// TwinCAT 3 PLC project PLC_Project
// ProgramVersion: 3.1.4024.0
// libraries:
//   Tc2_MC2, * (Beckhoff Automation GmbH)
//   Tc2_Standard, * (Beckhoff Automation GmbH)
//   Tc2_System, * (Beckhoff Automation GmbH)
//   Tc3_Module, * (Beckhoff Automation GmbH)
//   VisuSymbols,3.5.10.0,System
// project tree:
//   / GlobalTextList.TcGTLO, PlcTask.TcTTO, Visualization Manager.TcVMO (not stored), VISU_TASK.TcTTO
//   GVLs/ GVL_VARS1.TcGVL, GVL_VARS2.TcGVL, GVL_VARS3.TcGVL, GVL_VARS4.TcGVL
//   POUs/ FB_Functions.TcPOU, MAIN.TcPOU
//   VISUs/ Screen1.TcVIS
// real-time tasks:
//   TASK PlcTask: cycle T#10ms, priority 20, ADS port 350
//   TASK VISU_TASK: cycle T#200000us, priority 30, ADS port 351
// motion (NC):
//   TASK NC-Project1 SAF: cycle T#2ms, priority 4, ADS port 501
//   TASK NC-Project1 SVB: cycle T#10ms, priority 8, ADS port 511
//   AXIS Axis 1 (id 1)
//     OtherSettings: AllowMotionCmdToSlave=true
//     encoder EncType=1
//     encoder EncId=129, EncType=1
//     drive DrvType=5
//       Analog: TorqueSetpointScale=10, ScaleFactorActTorque=0.1
//       TimeComp: TaskDelayCycles=1
//     controller CtrType=1
//       CtrPara: PriorControlFactor=1
//         Observer: BandWidth=20
//     controller CtrId=129, CtrType=1
//       CtrPara: PriorControlFactor=1
//         Observer: BandWidth=20
//   AXIS Axis 2 (id 2)
//     OtherSettings: AllowMotionCmdToSlave=true
//     encoder EncType=1
//     encoder EncId=130, EncType=1
//     drive DrvType=5
//       Analog: TorqueSetpointScale=10, ScaleFactorActTorque=0.1
//       TimeComp: TaskDelayCycles=1
//     controller CtrType=1
//       CtrPara: PriorControlFactor=1
//         Observer: BandWidth=20
//     controller CtrId=130, CtrType=1
//       CtrPara: PriorControlFactor=1
//         Observer: BandWidth=20
//   AXIS Axis 3 (id 3)
//     OtherSettings: AllowMotionCmdToSlave=true
//     encoder EncType=1
//     encoder EncId=131, EncType=1
//     drive DrvType=5
//       Analog: TorqueSetpointScale=10, ScaleFactorActTorque=0.1
//       TimeComp: TaskDelayCycles=1
//     controller CtrType=1
//       CtrPara: PriorControlFactor=1
//         Observer: BandWidth=20
//     controller CtrId=131, CtrType=1
//       CtrPara: PriorControlFactor=1
//         Observer: BandWidth=20
//   AXIS Axis 4 (id 4)
//     OtherSettings: AllowMotionCmdToSlave=true
//     encoder EncType=1
//     encoder EncId=132, EncType=1
//     drive DrvType=5
//       Analog: TorqueSetpointScale=10, ScaleFactorActTorque=0.1
//       TimeComp: TaskDelayCycles=1
//     controller CtrType=1
//       CtrPara: PriorControlFactor=1
//         Observer: BandWidth=20
//     controller CtrId=132, CtrType=1
//       CtrPara: PriorControlFactor=1
//         Observer: BandWidth=20
// variable links:
//   PLC-Project/PLC-Project Instance <-> NC-Project1 SAF/Axes/Axis 1
//     PlcTask Inputs/MAIN.Axis[0][0].NcToPlc <-> Outputs/ToPlc
//     PlcTask Inputs/MAIN.Axis[0][1].NcToPlc <-> Outputs/ToPlc2
//     PlcTask Outputs/MAIN.Axis[0][0].PlcToNc <-> Inputs/FromPlc
//     PlcTask Outputs/MAIN.Axis[0][1].PlcToNc <-> Inputs/FromPlc2
//   PLC-Project/PLC-Project Instance <-> NC-Project1 SAF/Axes/Axis 2
//     PlcTask Inputs/MAIN.Axis[1][0].NcToPlc <-> Outputs/ToPlc
//     PlcTask Inputs/MAIN.Axis[1][1].NcToPlc <-> Outputs/ToPlc2
//     PlcTask Outputs/MAIN.Axis[1][0].PlcToNc <-> Inputs/FromPlc
//     PlcTask Outputs/MAIN.Axis[1][1].PlcToNc <-> Inputs/FromPlc2
//   PLC-Project/PLC-Project Instance <-> NC-Project1 SAF/Axes/Axis 3
//     PlcTask Inputs/MAIN.Axis[2][0].NcToPlc <-> Outputs/ToPlc
//     PlcTask Inputs/MAIN.Axis[2][1].NcToPlc <-> Outputs/ToPlc2
//     PlcTask Outputs/MAIN.Axis[2][0].PlcToNc <-> Inputs/FromPlc
//     PlcTask Outputs/MAIN.Axis[2][1].PlcToNc <-> Inputs/FromPlc2
//   PLC-Project/PLC-Project Instance <-> NC-Project1 SAF/Axes/Axis 4
//     PlcTask Inputs/MAIN.Axis[3][0].NcToPlc <-> Outputs/ToPlc
//     PlcTask Inputs/MAIN.Axis[3][1].NcToPlc <-> Outputs/ToPlc2
//     PlcTask Outputs/MAIN.Axis[3][0].PlcToNc <-> Inputs/FromPlc
//     PlcTask Outputs/MAIN.Axis[3][1].PlcToNc <-> Inputs/FromPlc2

CONFIGURATION PLC_Project
    RESOURCE PLC ON TwinCAT3
        TASK PlcTask(INTERVAL := T#10ms, PRIORITY := 20);
        TASK VISU_TASK(INTERVAL := T#200000us, PRIORITY := 30);
        PROGRAM MAIN WITH PlcTask : MAIN;
        PROGRAM VisuElems_Visu_Prg WITH VISU_TASK : VisuElems.Visu_Prg;
    END_RESOURCE
END_CONFIGURATION

// ---- GVLs/GVL_VARS1.TcGVL
{attribute 'qualified_only'}
VAR_GLOBAL
	position: UINT := 0;
	velocity: UINT := 0;
	acceleration: UINT := 0;
	execute: BOOL := FALSE;
END_VAR

// ---- GVLs/GVL_VARS2.TcGVL
{attribute 'qualified_only'}
VAR_GLOBAL
	position: UINT := 0;
	velocity: UINT := 0;
	acceleration: UINT := 0;
	execute: BOOL := FALSE;
END_VAR

// ---- GVLs/GVL_VARS3.TcGVL
{attribute 'qualified_only'}
VAR_GLOBAL
	position: UINT := 0;
	velocity: UINT := 0;
	acceleration: UINT := 0;
	execute: BOOL := FALSE;
END_VAR

// ---- GVLs/GVL_VARS4.TcGVL
{attribute 'qualified_only'}
VAR_GLOBAL
	position: UINT := 0;
	velocity: UINT := 0;
	acceleration: UINT := 0;
	execute: BOOL := FALSE;
END_VAR

// ---- POUs/MAIN.TcPOU
PROGRAM MAIN
VAR
	//nState: UINT := 0;
	Axis : ARRAY [0..3] OF ARRAY [0..1] OF AXIS_REF;
	MoveAbsolute : MC_MoveAbsolute;
	MoveRelative : MC_MoveRelative;
	WriteParameter : MC_WriteParameter;
	ReadParameter : MC_ReadParameter;
	AxisPower : MC_Power;
	Reset : MC_Reset;
	FB_Functions : FB_Functions;
	AxisParams : MC_AxisParameter;
	ReadDriveAddress : MC_ReadDriveAddress;
	SetControlLoop : MC_SelectControlLoop;
	ReadBoolParameter : MC_ReadBoolParameter;
	WriteBoolParameter : MC_WriteBoolParameter;
	Axis1LoopID : UINT;
	Axis2LoopID : UINT;
	Axis3LoopID : UINT;
	Axis4LoopID : UINT;
END_VAR

//Axis1[0]();
//Axis1[1]();
//Axis1[2]();
//Axis1();

Axis[0][0](); // incremental encoder axis 1
Axis[0][1](); // absolute encoder axis 1
Axis1LoopID := Axis[0][0].NcToPlc.ActiveControlLoopIndex;

Axis[1][0](); // incremental encoder axis 2
Axis[1][1](); // absolute encoder axis 2
Axis2LoopID := Axis[1][0].NcToPlc.ActiveControlLoopIndex;

Axis[2][0](); // incremental encoder axis 3
Axis[2][1](); // absolute encoder axis 3
Axis3LoopID := Axis[2][0].NcToPlc.ActiveControlLoopIndex;

Axis[3][0](); // incremental encoder axis 4
Axis[3][1](); // absolute encoder axis 4
Axis4LoopID := Axis[3][0].NcToPlc.ActiveControlLoopIndex;



//E_NcEncoderType.NcEncoderType_Simulation

//CASE nState OF
//	0:
//	nState := 10;
//	
//	10:
//	MoveAbsolute(Axis:=Axis1[0],Execute:=FALSE);
//	Reset(Axis:=Axis1[0],Execute:=FALSE);
//	nState := 20;
//	
//	20:
//	AxisPower(Axis:=Axis1[0],
//			Enable:=TRUE,
//			Enable_Positive:=TRUE,
//			Enable_Negative:=TRUE);
//			
//	IF GVL_VARS1.execute THEN
//		nState := 30;
//	END_IF
//
//	
//	30:
//	MoveAbsolute(Axis:=Axis1[0],
//					Position:=GVL_VARS1.position,
//					Velocity:=GVL_VARS1.velocity);
//	MoveAbsolute(Axis:=Axis1[0],
//					Execute:=TRUE);		
//	IF MoveAbsolute.Done THEN
//		MoveAbsolute(Axis:=Axis1[0],Execute:=FALSE);
//	END_IF
//	GVL_VARS1.execute := FALSE;
//	nState := 10;
//END_CASE


//AxisPower(Axis:=Axis1);
//MoveAbsolute(Axis:=Axis1);
//Reset(Axis:=Axis1);

END_PROGRAM

// ---- POUs/FB_Functions.TcPOU
FUNCTION_BLOCK FB_Functions
VAR_INPUT
END_VAR
VAR_OUTPUT
END_VAR
VAR
END_VAR

{attribute 'TcRpcEnable'}
METHOD M_EnableAxis : BOOL
VAR_INPUT
	axisID : UINT;
	loopID : UINT;
END_VAR
Main.AxisPower(Axis:=Main.Axis[axisID][loopID],Enable:=TRUE,Enable_Positive:=TRUE,Enable_Negative:=TRUE); 

RETURN;
END_METHOD

{attribute 'TcRpcEnable'}
METHOD M_MoveAbsolute : BOOL
VAR_INPUT
	axisID : UINT;
	loopID : UINT;
	position : LREAL;
	velocity : LREAL;
END_VAR
Main.AxisPower(Axis:=Main.Axis[axisID][loopID],Enable:=TRUE,Enable_Positive:=TRUE,Enable_Negative:=TRUE); 

WHILE Main.Axis[axisID][loopID].Status.Operational = FALSE DO
	Main.MoveAbsolute(Axis:=Main.Axis[axisID][loopID],Execute:=FALSE);
END_WHILE

Main.MoveAbsolute(Axis:=Main.Axis[axisID][loopID],Execute:=FALSE);
Main.Reset(Axis:=Main.Axis[axisID][loopID],Execute:=FALSE);
			
Main.MoveAbsolute(Axis:=main.Axis[axisID][loopID],Position:=position,Velocity:=velocity);
					
Main.MoveAbsolute(Axis:=Main.Axis[axisID][loopID],Execute:=TRUE);

Main.MoveAbsolute(Axis:=Main.Axis[axisID][loopID],Execute:=FALSE);

RETURN;
END_METHOD

{attribute 'TcRpcEnable'}
METHOD M_MoveHome : BOOL
VAR_INPUT
	axisID : UINT;
	loopID : UINT;
END_VAR
Main.AxisPower(Axis:=Main.Axis[axisID][loopID],Enable:=TRUE,Enable_Positive:=TRUE,Enable_Negative:=TRUE); 

WHILE Main.Axis[axisID][loopID].Status.Operational = FALSE DO
	Main.MoveHome(Axis:=Main.Axis[axisID][loopID],Execute:=FALSE);
END_WHILE

Main.MoveHome(Axis:=Main.Axis[axisID][loopID],Execute:=FALSE);
Main.Reset(Axis:=Main.Axis[axisID][loopID],Execute:=FALSE);

Main.MoveHome(Axis:=Main.Axis[axisID][loopID],Position:=0,HomingMode:=MC_DefaultHoming);

Main.MoveHome(Axis:=Main.Axis[axisID][loopID],Execute:=TRUE);

RETURN;
END_METHOD

{attribute 'TcRpcEnable'}
METHOD M_MoveRelative : BOOL
VAR_INPUT
	axisID : UINT;
	loopID : UINT;
	position : LREAL;
	velocity : LREAL;
END_VAR
Main.AxisPower(Axis:=Main.Axis[axisID][loopID],Enable:=TRUE,Enable_Positive:=TRUE,Enable_Negative:=TRUE); 

WHILE Main.Axis[axisID][loopID].Status.Operational = FALSE DO
	Main.MoveRelative(Axis:=Main.Axis[axisID][loopID],Execute:=FALSE);
END_WHILE

Main.MoveRelative(Axis:=Main.Axis[axisID][loopID],Execute:=FALSE);
Main.Reset(Axis:=Main.Axis[axisID][loopID],Execute:=FALSE);
			
Main.MoveRelative(Axis:=Main.Axis[axisID][loopID],Distance:=position,Velocity:=velocity);
					
Main.MoveRelative(Axis:=Main.Axis[axisID][loopID],Execute:=TRUE);

Main.MoveRelative(Axis:=Main.Axis[axisID][loopID],Execute:=FALSE);

RETURN;
END_METHOD

{attribute 'TcRpcEnable'}
METHOD M_ReadActiveLoop : UINT
VAR_INPUT
	axisID : UINT;
END_VAR
VAR_OUTPUT
	loopID : UINT;
END_VAR
loopID := Main.Axis[axisID][0].NcToPlc.ActiveControlLoopIndex;

RETURN;
END_METHOD

{attribute 'TcRpcEnable'}
METHOD M_ReadAxisMotion : LREAL
VAR_INPUT
	axisID : UINT;
END_VAR
VAR_OUTPUT
	position : LREAL;
	velocity : LREAL;
END_VAR
position := Main.Axis[axisID][0].NcToPlc.ActPos;

velocity := MAIN.Axis[axisID][0].NcToPlc.ActVelo;
END_METHOD

{attribute 'TcRpcEnable'}
METHOD M_ReadAxisParameters : LREAL
VAR_INPUT
	axisID : UINT;
	loopID : UINT;
END_VAR
VAR_OUTPUT
	maxVelocity : LREAL;
	maxAcceleration : LREAL;
	defaultAcceleration : LREAL;
	defaultJerk : LREAL;
	homingVelocity : LREAL;
	manualVelocityFast : LREAL;
	manualVelocitySlow : LREAL;
	jogIncrement : LREAL;
END_VAR
// Axis Max Velocity
Main.ReadParameter(Axis:=Main.Axis[axisID][loopID],ParameterNumber:=MC_AxisParameter.AxisMaxVelocity);
Main.ReadParameter(Axis:=Main.Axis[axisID][loopID],Enable:=TRUE);
WHILE Main.ReadParameter.Busy DO
	Main.ReadParameter(Axis:=Main.Axis[axisID][loopID],Enable:=FALSE);
END_WHILE
maxVelocity := Main.ReadParameter.Value;


// Axis Max Acceleration
Main.ReadParameter(Axis:=Main.Axis[axisID][loopID],ParameterNumber:=MC_AxisParameter.AxisMaximumAcceleration);
Main.ReadParameter(Axis:=Main.Axis[axisID][loopID],Enable:=TRUE);
WHILE Main.ReadParameter.Busy DO
	Main.ReadParameter(Axis:=Main.Axis[axisID][loopID],Enable:=FALSE);
END_WHILE
maxAcceleration := Main.ReadParameter.Value;


//Axis Default Acceleration
Main.ReadParameter(Axis:=Main.Axis[axisID][loopID],ParameterNumber:=MC_AxisParameter.AxisAcc);
Main.ReadParameter(Axis:=Main.Axis[axisID][loopID],Enable:=TRUE);
WHILE Main.ReadParameter.Busy DO
	Main.ReadParameter(Axis:=Main.Axis[axisID][loopID],Enable:=FALSE);
END_WHILE
defaultAcceleration := Main.ReadParameter.Value;


//Axis Default Jerk
Main.ReadParameter(Axis:=Main.Axis[axisID][loopID],ParameterNumber:=MC_AxisParameter.AxisJerk);
Main.ReadParameter(Axis:=Main.Axis[axisID][loopID],Enable:=TRUE);
WHILE Main.ReadParameter.Busy DO
	Main.ReadParameter(Axis:=Main.Axis[axisID][loopID],Enable:=FALSE);
END_WHILE
defaultJerk := Main.ReadParameter.Value;


//Axis Homing Velocity +ve direction
Main.ReadParameter(Axis:=Main.Axis[axisID][loopID],ParameterNumber:=MC_AxisParameter.AxisCalibrationVelocityForward);
Main.ReadParameter(Axis:=Main.Axis[axisID][loopID],Enable:=TRUE);
WHILE Main.ReadParameter.Busy DO
	Main.ReadParameter(Axis:=Main.Axis[axisID][loopID],Enable:=FALSE);
END_WHILE
homingVelocity := Main.ReadParameter.Value;


//Axis Manual Velocity (Fast)
Main.ReadParameter(Axis:=Main.Axis[axisID][loopID],ParameterNumber:=MC_AxisParameter.AxisManualVelocityFast);
Main.ReadParameter(Axis:=Main.Axis[axisID][loopID],Enable:=TRUE);
WHILE Main.ReadParameter.Busy DO
	Main.ReadParameter(Axis:=Main.Axis[axisID][loopID],Enable:=FALSE);
END_WHILE
manualVelocityFast := Main.ReadParameter.Value;


//Axis Manual Velocity (Slow)
Main.ReadParameter(Axis:=Main.Axis[axisID][loopID],ParameterNumber:=MC_AxisParameter.AxisManualVelocitySlow);
Main.ReadParameter(Axis:=Main.Axis[axisID][loopID],Enable:=TRUE);
WHILE Main.ReadParameter.Busy DO
	Main.ReadParameter(Axis:=Main.Axis[axisID][loopID],Enable:=FALSE);
END_WHILE
manualVelocitySlow := Main.ReadParameter.Value;


//Axis Jog Increment +ve Direction
Main.ReadParameter(Axis:=Main.Axis[axisID][loopID],ParameterNumber:=MC_AxisParameter.AxisJogIncrementForward);
Main.ReadParameter(Axis:=Main.Axis[axisID][loopID],Enable:=TRUE);
WHILE Main.ReadParameter.Busy DO
	Main.ReadParameter(Axis:=Main.Axis[axisID][loopID],Enable:=FALSE);
END_WHILE
jogIncrement := Main.ReadParameter.Value;

RETURN;
END_METHOD

{attribute 'TcRpcEnable'}
METHOD M_ReadControllerParameters : UINT
VAR_INPUT
	axisID : UINT;
	loopID : UINT;
END_VAR
VAR_OUTPUT
	kvParam : LREAL;
END_VAR
// Controller Kv parameter
Main.ReadParameter(Axis:=Main.Axis[axisID][loopID],ParameterNumber:=MC_AxisParameter.AxisPositionControlKv);
Main.ReadParameter(Axis:=Main.Axis[axisID][loopID],Enable:=TRUE);
WHILE Main.ReadParameter.Busy DO
	Main.ReadParameter(Axis:=Main.Axis[axisID][loopID],Enable:=FALSE);
END_WHILE
kvParam := Main.ReadParameter.Value;
RETURN;
END_METHOD

{attribute 'TcRpcEnable'}
METHOD M_ReadDriveParameters : BOOL
VAR_INPUT
	axisID : UINT;
	loopID : UINT;
END_VAR
VAR_OUTPUT
	inversePolarity : BOOL;
	refVelocity : LREAL;
END_VAR
// Drive inverse motor polarity
Main.ReadBoolParameter(Axis:=Main.Axis[axisID][loopID],ParameterNumber:=MC_AxisParameter.AxisMotorDirectionInverse,Enable:=TRUE,ReadMode:=E_ReadMode.READMODE_ONCE);
//Main.ReadBoolParameter(Axis:=Main.Axis[axisID][loopID],Enable:=TRUE);
//WHILE (Main.ReadBoolParameter.Busy = TRUE) DO
//	Main.ReadBoolParameter(Axis:=Main.Axis[axisID][loopID],Enable:=FALSE);
//END_WHILE
//IF Main.ReadBoolParameter.Valid THEN
	inversePolarity := Main.ReadBoolParameter.Value;
//END_IF
Main.ReadBoolParameter(Axis:=Main.Axis[axisID][loopID],Enable:=FALSE);

// Drive Reference Velocity
Main.ReadParameter(Axis:=Main.Axis[axisID][loopID],ParameterNumber:=MC_AxisParameter.AxisRefVeloOnRefOutput);
Main.ReadParameter(Axis:=Main.Axis[axisID][loopID],Enable:=TRUE);
WHILE Main.ReadParameter.Busy DO
	Main.ReadParameter(Axis:=Main.Axis[axisID][loopID],Enable:=FALSE);
END_WHILE
refVelocity := Main.ReadParameter.Value;

RETURN;
END_METHOD

{attribute 'TcRpcEnable'}
METHOD M_ReadEncoderParameters : UINT
VAR_INPUT
	axisID : UINT;
	loopID : UINT;
END_VAR
VAR_OUTPUT
	invertEncoderDirection : BOOL;
	scalingFactorNumerator : LREAL;
	scalingFactorDenominator : LREAL;
	encoderOffset : LREAL;
	encoderMask : LREAL;
END_VAR
// Invert Encoder Direction
Main.ReadBoolParameter(Axis:=Main.Axis[axisID][loopID],ParameterNumber:=MC_AxisParameter.AxisEncoderDirectionInverse,Enable:=TRUE,ReadMode:=E_ReadMode.READMODE_ONCE);
//Main.ReadBoolParameter(Axis:=Main.Axis[axisID][loopID]);
//WHILE (Main.ReadParameter.Busy = TRUE) DO
//	Main.ReadBoolParameter(Axis:=Main.Axis[axisID][loopID],Enable:=FALSE);
//END_WHILE
//IF Main.ReadBoolParameter.Valid THEN
	invertEncoderDirection := Main.ReadBoolParameter.Value;
//END_IF
Main.ReadBoolParameter(Axis:=Main.Axis[axisID][loopID],Enable:=FALSE);


// Encoder Scaling Factor Numerator
Main.ReadParameter(Axis:=Main.Axis[axisID][loopID],ParameterNumber:=MC_AxisParameter.AxisEncoderScalingNumerator);
Main.ReadParameter(Axis:=Main.Axis[axisID][loopID],Enable:=TRUE);
WHILE Main.ReadParameter.Busy DO
	Main.ReadParameter(Axis:=Main.Axis[axisID][loopID],Enable:=FALSE);
END_WHILE
scalingFactorNumerator := Main.ReadParameter.Value;


// Encoder Scaling Factor Denominator
Main.ReadParameter(Axis:=Main.Axis[axisID][loopID],ParameterNumber:=MC_AxisParameter.AxisEncoderScalingDenominator);
Main.ReadParameter(Axis:=Main.Axis[axisID][loopID],Enable:=TRUE);
WHILE Main.ReadParameter.Busy DO
	Main.ReadParameter(Axis:=Main.Axis[axisID][loopID],Enable:=FALSE);
END_WHILE
scalingFactorDenominator := Main.ReadParameter.Value;


// Encoder Offset
Main.ReadParameter(Axis:=Main.Axis[axisID][loopID],ParameterNumber:=MC_AxisParameter.AxisEncoderOffset);
Main.ReadParameter(Axis:=Main.Axis[axisID][loopID],Enable:=TRUE);
WHILE Main.ReadParameter.Busy DO
	Main.ReadParameter(Axis:=Main.Axis[axisID][loopID],Enable:=FALSE);
END_WHILE
encoderOffset := Main.ReadParameter.Value;


// Encoder Mask
Main.ReadParameter(Axis:=Main.Axis[axisID][loopID],ParameterNumber:=MC_AxisParameter.AxisEncoderMask);
Main.ReadParameter(Axis:=Main.Axis[axisID][loopID],Enable:=TRUE);
WHILE Main.ReadParameter.Busy DO
	Main.ReadParameter(Axis:=Main.Axis[axisID][loopID],Enable:=FALSE);
END_WHILE
encoderMask := Main.ReadParameter.Value;


RETURN;
END_METHOD

{attribute 'TcRpcEnable'}
METHOD M_SetActiveEncoder : BOOL
VAR_INPUT
	axisID : UINT;
	loopID : UINT;
END_VAR
Main.SetControlLoop(Axis:=Main.Axis[axisID][loopID],Execute:=FALSE,SelectType:=E_SelectControlLoopType.SelectControlLoopType_Standard,EncoderIndex:=loopID);
Main.SetControlLoop(Axis:=Main.Axis[axisID][loopID],Execute:=TRUE);
WHILE (Main.SetControlLoop.Done=FALSE) DO
	Main.SetControlLoop(Axis:=Main.Axis[axisID][loopID],Execute:=FALSE);
END_WHILE

RETURN;
END_METHOD

{attribute 'TcRpcEnable'}
METHOD M_SetActualPosition : BOOL
VAR_INPUT
	axisID : UINT;
	loopID : UINT;
	position : LREAL;
END_VAR
Main.SetActualPosition(Axis:=Main.Axis[axisID][loopID],Position:=position,Mode:=FALSE,Execute:=FALSE);
Main.SetActualPosition(Axis:=Main.Axis[axisID][loopID],Execute:=TRUE);
WHILE (Main.SetActualPosition.Done=FALSE) DO
	Main.SetActualPosition(Axis:=Main.Axis[axisID][loopID],Execute:=FALSE);
END_WHILE

RETURN;
END_METHOD

{attribute 'TcRpcEnable'}
METHOD M_WriteAxisParameters : BOOL
VAR_INPUT
	axisID: UINT;
	loopID: UINT;
	maxVelocity : LREAL;
	maxAcceleration : LREAL;
	defaultAcceleration : LREAL;
	defaultJerk : LREAL;
	homingVelocity : LREAL;
	manualVelocityFast : LREAL;
	manualVelocitySlow : LREAL;
	jogIncrement : LREAL;
END_VAR
// Axis Max Velocity
Main.WriteParameter(Axis:=Main.Axis[axisID][loopID],ParameterNumber:=MC_AxisParameter.AxisMaxVelocity,Value:=maxVelocity);
Main.WriteParameter(Axis:=Main.Axis[axisID][loopID],Execute:=TRUE);
WHILE (Main.WriteParameter.Busy) DO
	Main.WriteParameter(Axis:=Main.Axis[axisID][loopID],Execute:=FALSE);
END_WHILE

// Axis Max Acceleration
Main.WriteParameter(Axis:=Main.Axis[axisID][loopID],ParameterNumber:=MC_AxisParameter.AxisMaximumAcceleration,Value:=maxAcceleration);
Main.WriteParameter(Axis:=Main.Axis[axisID][loopID],Execute:=TRUE);
WHILE (Main.WriteParameter.Busy) DO
	Main.WriteParameter(Axis:=Main.Axis[axisID][loopID],Execute:=FALSE);
END_WHILE

//Axis Max Deceleration
Main.WriteParameter(Axis:=Main.Axis[axisID][loopID],ParameterNumber:=MC_AxisParameter.AxisMaximumDeceleration,Value:=maxAcceleration);
Main.WriteParameter(Axis:=Main.Axis[axisID][loopID],Execute:=TRUE);
WHILE (Main.WriteParameter.Busy) DO
	Main.WriteParameter(Axis:=Main.Axis[axisID][loopID],Execute:=FALSE);
END_WHILE

//Axis Default Acceleration
Main.WriteParameter(Axis:=Main.Axis[axisID][loopID],ParameterNumber:=MC_AxisParameter.AxisAcc,Value:=defaultAcceleration);
Main.WriteParameter(Axis:=Main.Axis[axisID][loopID],Execute:=TRUE);
WHILE (Main.WriteParameter.Busy) DO
	Main.WriteParameter(Axis:=Main.Axis[axisID][loopID],Execute:=FALSE);
END_WHILE

//Axis Default Deceleration
Main.WriteParameter(Axis:=Main.Axis[axisID][loopID],ParameterNumber:=MC_AxisParameter.AxisDec,Value:=defaultAcceleration);
Main.WriteParameter(Axis:=Main.Axis[axisID][loopID],Execute:=TRUE);
WHILE (Main.WriteParameter.Busy) DO
	Main.WriteParameter(Axis:=Main.Axis[axisID][loopID],Execute:=FALSE);
END_WHILE

//Axis Default Jerk
Main.WriteParameter(Axis:=Main.Axis[axisID][loopID],ParameterNumber:=MC_AxisParameter.AxisJerk,Value:=defaultJerk);
Main.WriteParameter(Axis:=Main.Axis[axisID][loopID],Execute:=TRUE);
WHILE (Main.WriteParameter.Busy) DO
	Main.WriteParameter(Axis:=Main.Axis[axisID][loopID],Execute:=FALSE);
END_WHILE

//Axis Homing Velocity +ve direction
Main.WriteParameter(Axis:=Main.Axis[axisID][loopID],ParameterNumber:=MC_AxisParameter.AxisCalibrationVelocityForward,Value:=homingVelocity);
Main.WriteParameter(Axis:=Main.Axis[axisID][loopID],Execute:=TRUE);
WHILE (Main.WriteParameter.Busy) DO
	Main.WriteParameter(Axis:=Main.Axis[axisID][loopID],Execute:=FALSE);
END_WHILE

//Axis Homing Velocity -ve Direction
Main.WriteParameter(Axis:=Main.Axis[axisID][loopID],ParameterNumber:=MC_AxisParameter.AxisCalibrationVelocityBackward,Value:=homingVelocity);
Main.WriteParameter(Axis:=Main.Axis[axisID][loopID],Execute:=TRUE);
WHILE (Main.WriteParameter.Busy) DO
	Main.WriteParameter(Axis:=Main.Axis[axisID][loopID],Execute:=FALSE);
END_WHILE

//Axis Manual Velocity (Fast)
Main.WriteParameter(Axis:=Main.Axis[axisID][loopID],ParameterNumber:=MC_AxisParameter.AxisManualVelocityFast,Value:=manualVelocityFast);
Main.WriteParameter(Axis:=Main.Axis[axisID][loopID],Execute:=TRUE);
WHILE (Main.WriteParameter.Busy) DO
	Main.WriteParameter(Axis:=Main.Axis[axisID][loopID],Execute:=FALSE);
END_WHILE

//Axis Manual Velocity (Slow)
Main.WriteParameter(Axis:=Main.Axis[axisID][loopID],ParameterNumber:=MC_AxisParameter.AxisManualVelocitySlow,Value:=manualVelocitySlow);
Main.WriteParameter(Axis:=Main.Axis[axisID][loopID],Execute:=TRUE);
WHILE (Main.WriteParameter.Busy) DO
	Main.WriteParameter(Axis:=Main.Axis[axisID][loopID],Execute:=FALSE);
END_WHILE

//Axis Jog Increment +ve Direction
Main.WriteParameter(Axis:=Main.Axis[axisID][loopID],ParameterNumber:=MC_AxisParameter.AxisJogIncrementForward,Value:=jogIncrement);
Main.WriteParameter(Axis:=Main.Axis[axisID][loopID],Execute:=TRUE);
WHILE (Main.WriteParameter.Busy) DO
	Main.WriteParameter(Axis:=Main.Axis[axisID][loopID],Execute:=FALSE);
END_WHILE

//Axis Jog Increment -ve Direction
Main.WriteParameter(Axis:=Main.Axis[axisID][loopID],ParameterNumber:=MC_AxisParameter.AxisJogIncrementBackward,Value:=jogIncrement);
Main.WriteParameter(Axis:=Main.Axis[axisID][loopID],Execute:=TRUE);
WHILE (Main.WriteParameter.Busy) DO
	Main.WriteParameter(Axis:=Main.Axis[axisID][loopID],Execute:=FALSE);
END_WHILE

RETURN;
END_METHOD

{attribute 'TcRpcEnable'}
METHOD M_WriteControllerParameters : BOOL
VAR_INPUT
	axisID : UINT;
	loopID : UINT;
	kvParam : LREAL;
END_VAR
// Controller Kv Parameter
Main.WriteParameter(Axis:=Main.Axis[axisID][loopID],ParameterNumber:=MC_AxisParameter.AxisPositionControlKv,Value:=kvParam);
Main.WriteParameter(Axis:=Main.Axis[axisID][loopID],Execute:=TRUE);
WHILE (Main.WriteParameter.Busy) DO
	Main.WriteParameter(Axis:=Main.Axis[axisID][loopID],Execute:=FALSE);
END_WHILE
END_METHOD

{attribute 'TcRpcEnable'}
METHOD M_WriteDriveParameters : BOOL
VAR_INPUT
	axisID : UINT;
	loopID : UINT;
	invertPolarity : BOOL;
	refVelocity : LREAL;
END_VAR
// Inverse motor polarity
Main.WriteBoolParameter(Axis:=Main.Axis[axisID][loopID],ParameterNumber:=MC_AxisParameter.AxisMotorDirectionInverse,Value:=invertPolarity);
Main.WriteBoolParameter(Axis:=Main.Axis[axisID][loopID],Execute:=TRUE);
WHILE (Main.WriteBoolParameter.Busy) DO
	Main.WriteBoolParameter(Axis:=Main.Axis[axisID][loopID],Execute:=FALSE);
END_WHILE
Main.WriteBoolParameter(Axis:=Main.Axis[axisID][loopID],Execute:=FALSE);

// Drive Reference Velocity
Main.WriteParameter(Axis:=Main.Axis[axisID][loopID],ParameterNumber:=MC_AxisParameter.AxisRefVeloOnRefOutput,Value:=refVelocity);
Main.WriteParameter(Axis:=Main.Axis[axisID][loopID],Execute:=TRUE);
WHILE (Main.WriteParameter.Busy) DO
	Main.WriteParameter(Axis:=Main.Axis[axisID][loopID],Execute:=FALSE);
END_WHILE
END_METHOD

{attribute 'TcRpcEnable'}
METHOD M_WriteEncoderParameters : BOOL
VAR_INPUT
	axisID : UINT;
	loopID : UINT;
	invertEncoderDirection : BOOL;
	scalingFactorNumerator : LREAL;
	scalingFactorDenominator : LREAL;
	encoderOffset : LREAL;
	encoderMask : DINT;
END_VAR
// Encoder direction inverse
Main.WriteBoolParameter(Axis:=Main.Axis[axisID][loopID],ParameterNumber:=MC_AxisParameter.AxisEncoderDirectionInverse,Value:=invertEncoderDirection);
Main.WriteBoolParameter(Axis:=Main.Axis[axisID][loopID],Execute:=TRUE);
WHILE (Main.WriteBoolParameter.Busy) DO
	Main.WriteBoolParameter(Axis:=Main.Axis[axisID][loopID],Execute:=FALSE);
END_WHILE
Main.WriteBoolParameter(Axis:=Main.Axis[axisID][loopID],Execute:=FALSE);

// Encoder scaling factor numerator
Main.WriteParameter(Axis:=Main.Axis[axisID][loopID],ParameterNumber:=MC_AxisParameter.AxisEncoderScalingNumerator,Value:=scalingFactorNumerator);
Main.WriteParameter(Axis:=Main.Axis[axisID][loopID],Execute:=TRUE);
WHILE (Main.WriteParameter.Busy) DO
	Main.WriteParameter(Axis:=Main.Axis[axisID][loopID],Execute:=FALSE);
END_WHILE

// Encoder scaling factor denominator
Main.WriteParameter(Axis:=Main.Axis[axisID][loopID],ParameterNumber:=MC_AxisParameter.AxisEncoderScalingDenominator,Value:=scalingFactorDenominator);
Main.WriteParameter(Axis:=Main.Axis[axisID][loopID],Execute:=TRUE);
WHILE (Main.WriteParameter.Busy) DO
	Main.WriteParameter(Axis:=Main.Axis[axisID][loopID],Execute:=FALSE);
END_WHILE

// Encoder offset
Main.WriteParameter(Axis:=Main.Axis[axisID][loopID],ParameterNumber:=MC_AxisParameter.AxisEncoderOffset,Value:=encoderOffset);
Main.WriteParameter(Axis:=Main.Axis[axisID][loopID],Execute:=TRUE);
WHILE (Main.WriteParameter.Busy) DO
	Main.WriteParameter(Axis:=Main.Axis[axisID][loopID],Execute:=FALSE);
END_WHILE

// Encoder Mask
Main.WriteParameter(Axis:=Main.Axis[axisID][loopID],ParameterNumber:=MC_AxisParameter.AxisEncoderMask,Value:=encoderMask);
Main.WriteParameter(Axis:=Main.Axis[axisID][loopID],Execute:=TRUE);
WHILE (Main.WriteParameter.Busy) DO
	Main.WriteParameter(Axis:=Main.Axis[axisID][loopID],Execute:=FALSE);
END_WHILE

RETURN;
END_METHOD

END_FUNCTION_BLOCK

// ---- GlobalTextList.TcGTLO
TEXTLIST GlobalTextList
  600 = '%4.3f'
  13 = '%i'
  301 = '%s'
  702 = 'Active control loop:'
  64 = 'Actual Position'
  16 = 'Actual velocity'
  0 = 'Axis 1'
  151 = 'Axis 2'
  802 = 'Axis 3'
  955 = 'Axis 4'
  110 = 'Error'
  199 = 'Error ID'
  558 = 'In target position'
  541 = 'In target position:'
  510 = 'Moving'
  389 = 'Moving:'
  537 = 'Reset'
  12 = 'Set Position'
  587 = 'Standstill:'
END_TEXTLIST

// ---- VISUs/Screen1.TcVIS
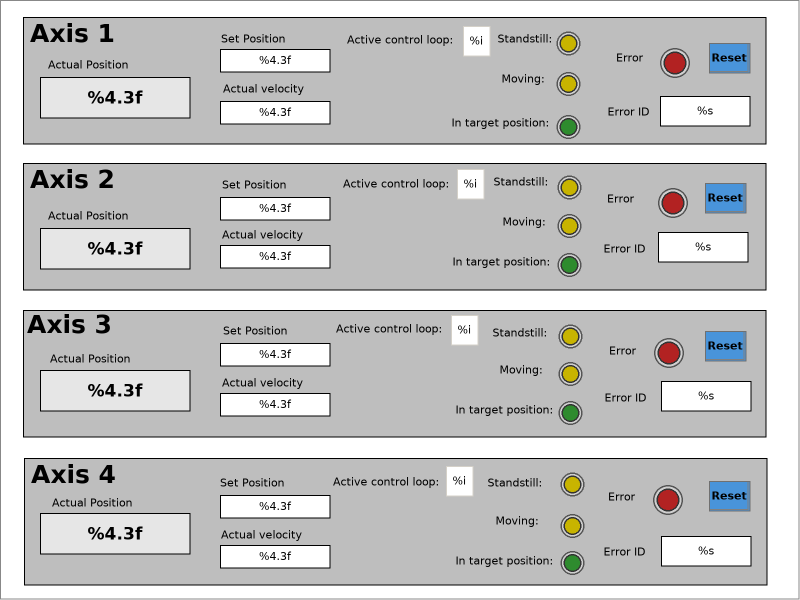
VISUALIZATION Screen1  // 800x600
    Rectangle (23,17 743x127)
    Rectangle (23,163 743x127)
    Rectangle (23,310 743x127)
    Rectangle (24,458 743x127)
    Label (27,18 110x30), "Axis 1"
    Label (27,164 110x30), "Axis 2"
    Label (24,309 110x30), "Axis 3"
    Label (28,459 110x30), "Axis 4"
    Textfield (40,77 150x41), "%4.3f", text variable: MAIN.Axis[0][MAIN.Axis1LoopID].NcToPlc.ActPos
    Label (45,50 150x30), "Actual Position"
    Label (45,201 150x30), "Actual Position"
    Label (47,344 150x30), "Actual Position"
    Label (49,488 150x30), "Actual Position"
    Textfield (40,228 150x41), "%4.3f", text variable: MAIN.Axis[1][MAIN.Axis2LoopID].NcToPlc.ActPos
    Textfield (40,370 150x41), "%4.3f", text variable: MAIN.Axis[2][MAIN.Axis3LoopID].NcToPlc.ActPos
    Textfield (40,513 150x41), "%4.3f", text variable: MAIN.Axis[3][MAIN.Axis4LoopID].NcToPlc.ActPos
    Label (218,24 150x30), "Set Position"
    Lamp1 (658,42 34x42), variable: MAIN.Axis[0][MAIN.Axis1LoopID].Status.Error, style: Lamp-Lamp1-Red
    Label (610,43 39x30), "Error"
    Label (596,97 65x30), "Error ID"
    Textfield (660,96 90x30), "%s", text variable: MAIN.Axis[0][MAIN.Axis1LoopID].Status.ErrorID
    Textfield (220,49 110x23), "%4.3f", text variable: MAIN.Axis[0][MAIN.Axis1LoopID].NcToPlc.TargetPos
    Textfield (220,101 110x23), "%4.3f", text variable: MAIN.Axis[0][MAIN.Axis1LoopID].NcToPlc.ActVelo
    Label (220,74 150x30), "Actual velocity"
    Label (219,170 150x30), "Set Position"
    Label (220,316 150x30), "Set Position"
    Label (217,468 150x30), "Set Position"
    Textfield (220,197 110x23), "%4.3f", text variable: MAIN.Axis[1][MAIN.Axis2LoopID].NcToPlc.TargetPos
    Textfield (220,343 110x23), "%4.3f", text variable: MAIN.Axis[2][MAIN.Axis3LoopID].NcToPlc.TargetPos
    Textfield (220,495 110x23), "%4.3f", text variable: MAIN.Axis[3][MAIN.Axis4LoopID].NcToPlc.TargetPos
    Label (219,220 150x30), "Actual velocity"
    Label (219,368 150x30), "Actual velocity"
    Label (218,520 150x30), "Actual velocity"
    Textfield (220,245 110x23), "%4.3f", text variable: MAIN.Axis[1][MAIN.Axis2LoopID].NcToPlc.ActVelo
    Textfield (220,393 110x23), "%4.3f", text variable: MAIN.Axis[3][MAIN.Axis3LoopID].NcToPlc.ActVelo
    Textfield (220,545 110x23), "%4.3f", text variable: MAIN.Axis[3][MAIN.Axis4LoopID].NcToPlc.ActVelo
    Label (601,184 39x30), "Error"
    Label (603,336 39x30), "Error"
    Label (602,482 39x30), "Error"
    Lamp1 (656,182 34x42), variable: MAIN.Axis[1][MAIN.Axis2LoopID].Status.Error, style: Lamp-Lamp1-Red
    Lamp1 (652,332 34x42), variable: MAIN.Axis[2][MAIN.Axis3LoopID].Status.Error, style: Lamp-Lamp1-Red
    Lamp1 (651,479 34x42), variable: MAIN.Axis[3][MAIN.Axis4LoopID].Status.Error, style: Lamp-Lamp1-Red
    Label (592,234 65x30), "Error ID"
    Label (593,383 65x30), "Error ID"
    Label (592,537 65x30), "Error ID"
    Textfield (658,232 90x30), "%s", text variable: MAIN.Axis[1][MAIN.Axis2LoopID].Status.ErrorID
    Textfield (661,381 90x30), "%s", text variable: MAIN.Axis[2][MAIN.Axis3LoopID].Status.ErrorID
    Textfield (661,536 90x30), "%s", text variable: MAIN.Axis[3][MAIN.Axis4LoopID].Status.ErrorID
    Lamp1 (555,67 27x34), variable: MAIN.Axis[0][MAIN.Axis1LoopID].Status.Moving, style: Lamp-Lamp1-Yellow
    Lamp1 (555,110 27x34), variable: MAIN.Axis[0][MAIN.Axis1LoopID].Status.InTargetPosition, style: Lamp-Lamp1-Green
    Label (491,24 68x30), "Standstill:"
    Label (450,108 101x30), "In target position:"
    Lamp1 (555,26 27x35), variable: MAIN.Axis[0][MAIN.Axis1LoopID].Status.StandStill, style: Lamp-Lamp1-Yellow
    Label (490,207 68x30), "Moving:"
    Lamp1 (556,170 27x35), variable: MAIN.Axis[1][MAIN.Axis2LoopID].Status.StandStill, style: Lamp-Lamp1-Yellow
    Lamp1 (556,209 27x34), variable: MAIN.Axis[1][MAIN.Axis2LoopID].Status.Moving, style: Lamp-Lamp1-Yellow
    Lamp1 (556,248 27x34), variable: MAIN.Axis[1][MAIN.Axis2LoopID].Status.InTargetPosition, style: Lamp-Lamp1-Green
    Lamp1 (559,467 27x35), variable: MAIN.Axis[3][MAIN.Axis4LoopID].Status.StandStill, style: Lamp-Lamp1-Yellow
    Lamp1 (557,319 27x35), variable: MAIN.Axis[2][MAIN.Axis3LoopID].Status.StandStill, style: Lamp-Lamp1-Yellow
    Lamp1 (557,357 27x34), variable: MAIN.Axis[2][MAIN.Axis3LoopID].Status.Moving, style: Lamp-Lamp1-Yellow
    Lamp1 (559,509 27x34), variable: MAIN.Axis[3][MAIN.Axis4LoopID].Status.Moving, style: Lamp-Lamp1-Yellow
    Lamp1 (557,396 27x34), variable: MAIN.Axis[2][MAIN.Axis3LoopID].Status.InTargetPosition, style: Lamp-Lamp1-Green
    Lamp1 (559,546 27x34), variable: MAIN.Axis[3][MAIN.Axis4LoopID].Status.InTargetPosition, style: Lamp-Lamp1-Green
    Label (487,167 68x30), "Standstill:"
    Label (486,318 68x30), "Standstill:"
    Label (481,468 68x30), "Standstill:"
    Label (489,64 68x30), "Moving:"
    Label (487,355 68x30), "Moving:"
    Label (483,506 68x30), "Moving:"
    Label (451,247 101x30), "In target position:"
    Label (454,395 101x30), "In target position:"
    Label (454,546 101x30), "In target position:"
    Label (342,25 116x30), "Active control loop:"
    Textfield (463,26 27x30), "%i", text variable: MAIN.Axis[0][0].NcToPlc.ActiveControlLoopIndex
    Textfield (457,169 27x30), "%i", text variable: MAIN.Axis[1][0].NcToPlc.ActiveControlLoopIndex
    Textfield (451,315 27x30), "%i", text variable: MAIN.Axis[2][0].NcToPlc.ActiveControlLoopIndex
    Textfield (446,466 27x30), "%i", text variable: MAIN.Axis[3][0].NcToPlc.ActiveControlLoopIndex
    Label (338,169 116x30), "Active control loop:"
    Label (331,314 116x30), "Active control loop:"
    Label (328,467 116x30), "Active control loop:"
    Button (709,43 41x30), "Reset"
        OnMouseDown: execute { MAIN.Reset(Axis:=MAIN.Axis[0][MAIN.Axis1LoopID],Execute:=TRUE); MAIN.Reset(Axis:=MAIN.Axis[0][MAIN.Axis1LoopID],Execute:=FALSE); }
    Button (705,183 41x30), "Reset"
        OnMouseDown: execute { MAIN.Reset(Axis:=MAIN.Axis[1][MAIN.Axis2LoopID],Execute:=TRUE); MAIN.Reset(Axis:=MAIN.Axis[1][MAIN.Axis2LoopID],Execute:=FALSE); }
    Button (705,331 41x30), "Reset"
        OnMouseDown: execute { MAIN.Reset(Axis:=MAIN.Axis[2][MAIN.Axis3LoopID],Execute:=TRUE); MAIN.Reset(Axis:=MAIN.Axis[2][MAIN.Axis3LoopID],Execute:=FALSE); }
    Button (709,481 41x30), "Reset"
        OnMouseDown: execute { MAIN.Reset(Axis:=MAIN.Axis[3][MAIN.Axis4LoopID],Execute:=TRUE); MAIN.Reset(Axis:=MAIN.Axis[3][MAIN.Axis4LoopID],Execute:=FALSE); }
END_VISUALIZATION
